Yaskawa INFORM job: R1B1.JBI

/JOB
//NAME R1B1
//POS
///NPOS 0,0,0,0,0,0
//INST
///DATE 2021/01/13 19:20
///ATTR SC,RW
///GROUP1 RB1,BS1
///LVARS 3,3,3,3,0,0,0,0
NOP
MOVJ P012 BP012 VJ=100.00 //P012

END
